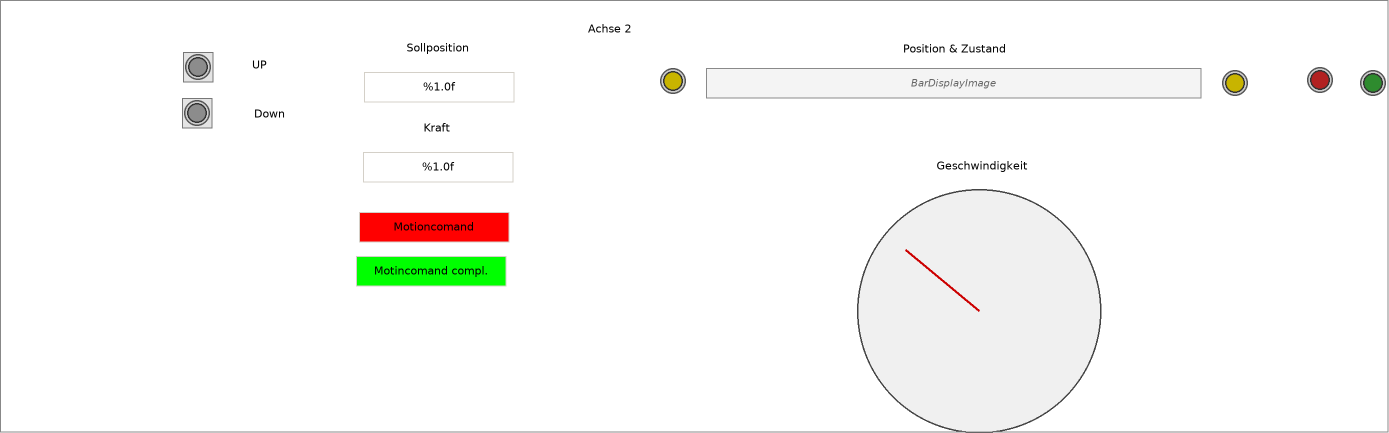
VISUALIZATION Visu_Achse2S_OLD  // 1389x433
    Label (859,34 191x30), "Position & Zustand"
    PushSwitch (182,52 32x30), variable: GVL.A2UP, behaviour: TAP, style: Switch-PushSwitch-Gray
    PushSwitch (181,98 32x30), variable: GVL.A2DOWN, behaviour: TAP, style: Switch-PushSwitch-Gray
    Label (225,50 69x30), "UP"
    Label (235,99 69x30), "Down"
    Textfield (364,72 150x30), "%1.0f", text variable: GVL.Eingabe_Sollposition_A2
    Label (363,33 150x30), "Sollposition"
    BarDisplayImage (706,68 495x30), value: GVL.ActualPosition_CYL2, style: BarDisplayImage-Gray, scale format: %.0f, scale 0..200
    Lamp1 (1304,65 32x30), variable: GVL.WarningActive_CYL2, style: Lamp-Lamp1-Red
    Lamp1 (1357,68 32x30), variable: GVL.Ready_CYL2, style: Lamp-Lamp1-Green
    Label (362,113 150x30), "Kraft"
    Textfield (363,152 150x30), "%1.0f", text variable: GVL.ActualForce_CYL2
    Label (907,151 150x30), "Geschwindigkeit"
    Meter360 (856,189 246x244), value: GVL.ActualSpeed_CYL2, style: Meter-Meter360-Gray, scale format: %.0f, scale -220..220
    Lamp1 (657,66 32x30), variable: GVL.LimitSwitchIn_CYL2, style: Lamp-Lamp1-Yellow
    Lamp1 (1219,68 32x30), variable: GVL.LimitSwitchOut_CYL2, style: Lamp-Lamp1-Yellow
    Textfield (356,256 150x30), "Motincomand compl.", text variable: GVL.ActualForce_CYL1, invisible if: GVL.MotionModeActive_CYL2
    Textfield (359,212 150x30), "Motioncomand", text variable: GVL.Eingabe_Sollposition_A1, invisible if: GVL.MotionCommandCompleted_CYL2
    Label (535,14 150x30), "Achse 2"
END_VISUALIZATION

(* stored: Version 1.1.0.1, ProductVersion 3.1.4024.12
   Visu Visu_Achse2S_OLD: Id {28911e40-3ff5-488a-9166-4871138dc69a} *)
